{attribute 'GeneratedUsingTerminal: EK1100-0000-0018'}
{attribute addProperty BoxType "EK1100-0000-0018"}
{attribute addProperty Id "Beckhoff_EPP2xxxEK1122Beckhoff_EPP2xxxEK1122_56176A052100"}
{attribute addProperty CRC "2396225124"}
{attribute addProperty Size "2100"}
TYPE Beckhoff_EPP2xxx_8ED37E64 EXTENDS EK1100_1FC0878B :
STRUCT
	{attribute addProperty Name "Beckhoff_EPP2xxxEK1122"}
	{attribute addProperty PreviousPort "Beckhoff EPP2xxx : B"}
	Beckhoff_EPP2xxxEK1122 : Beckhoff_EPP2xxxEK1122_56176A05;
END_STRUCT
END_TYPE

(* stored: Version 1.2.0.0, ProductVersion 3.1.4024.9
   DUT Beckhoff_EPP2xxx_8ED37E64: Id {894ede48-9f2f-4398-981d-41303573d625} *)
